// TwinCAT 3 PLC project Untitled1
// ProgramVersion: 3.1.4024.0
// libraries:
//   Tc2_MC2, * (Beckhoff Automation GmbH)
//   Tc2_Standard, * (Beckhoff Automation GmbH)
//   Tc2_System, * (Beckhoff Automation GmbH)
//   Tc3_Module, * (Beckhoff Automation GmbH)
// project tree:
//   / PlcTask.TcTTO
//   POUs/ MAIN.TcPOU, FB_PulseGenerate2s.TcPOU
// real-time tasks:
//   TASK PlcTask: cycle T#10ms, priority 20, ADS port 350
// motion (NC):
//   TASK NC-Task 1 SAF: cycle T#2ms, priority 4, ADS port 501
//   TASK NC-Task 1 SVB: cycle T#10ms, priority 8, ADS port 511
//   AXIS Axis 1 virtual (id 1)
//     OtherSettings: AllowMotionCmdToSlave=true
//     encoder EncType=1
//     drive DrvType=5
//       Analog: TorqueSetpointScale=10, ScaleFactorActTorque=0.1
//     controller CtrType=1
//       CtrPara: PriorControlFactor=1
//         Observer: BandWidth=20
// variable links:
//   Untitled1/Untitled1 Instance <-> NC-Task 1 SAF/Axes/Axis 1 virtual
//     PlcTask Inputs/MAIN.Axis1.NcToPlc <-> Outputs/ToPlc
//     PlcTask Outputs/MAIN.Axis1.PlcToNc <-> Inputs/FromPlc

CONFIGURATION Untitled1
    RESOURCE PLC ON TwinCAT3
        TASK PlcTask(INTERVAL := T#10ms, PRIORITY := 20);
        PROGRAM MAIN WITH PlcTask : MAIN;
    END_RESOURCE
END_CONFIGURATION

// ---- POUs/MAIN.TcPOU
PROGRAM MAIN
VAR
	/// axis reference data structure 
	Axis1: AXIS_REF;
END_VAR

METHOD ShiftRegister
VAR
	fbPulse : FB_PulseGenerate2s;	
	
	bStart: BOOL;
	
    nInByte  :  BYTE:=16#01; (*2#0100 0101*)   
    nVar : BYTE  := 1; 
	
	rt : R_TRIG;
	bSensor: BOOL;
	rtSensor : R_TRIG;
	
	rtCam1:R_TRIG;
	bCam1 : UINT;
END_VAR
fbPulse(bExcute:=bStart);

rt(CLK:=fbPulse.Q);
IF rt.Q THEN
	nInByte := SHL(nInByte,nVar);
END_IF

//register point
rtSensor(CLK:=bSensor);
IF rtSensor.Q THEN
	bSensor:= FALSE;
	nInByte := nInByte OR 16#01;
END_IF
//get bit at 9th position
rtCam1(CLK:=nInByte.3);
IF rtCam1.Q THEN
	bCam1:=bCam1+1;
END_IF
END_METHOD

END_PROGRAM

// ---- POUs/FB_PulseGenerate2s.TcPOU
FUNCTION_BLOCK FB_PulseGenerate2s
VAR_INPUT
	bExcute : BOOL;
END_VAR
VAR_OUTPUT
	Q	: BOOL;
END_VAR
VAR	
	rt : R_TRIG;
	ft : F_TRIG;
	tpT1	: TP;
	tonT1	: TON;
	tonT2	: TON;
	bEx1: BOOL;
	bEx2: BOOL;
END_VAR

rt(CLK:=bExcute);
ft(CLK:=bExcute);
//off function
IF ft.Q THEN
	bEx1 := FALSE;
	bEx2:=FALSE;
END_IF
tonT1(IN:=bEx1,PT:=T#1S) ;
tonT2(IN:=bEx2,PT:=T#1S) ;
//kích timer 1
IF 	rt.Q THEN
	bEx1:=TRUE ;
END_IF
//kích timer 2
IF tonT1.Q THEN
	bEx2:=TRUE;
	bEx1:= FALSE;
END_IF
IF tonT2.Q THEN
	bEx1 := TRUE;
	bEx2:=FALSE;
END_IF
//output
Q:=bEx1;

END_FUNCTION_BLOCK
